Fanuc TP program (LS listing): ground_truth.ls

/PROG  TOR_XL_LEARN_V6
/ATTR
OWNER		= MNEDITOR;
COMMENT		= "WeldPRO Auto-Gen";
PROG_SIZE	= 7125;
CREATE		= DATE 26-07-31  TIME 09:44:06;
MODIFIED	= DATE 26-07-31  TIME 10:09:20;
FILE_NAME	= TOR_XL_L;
VERSION		= 0;
LINE_COUNT	= 113;
MEMORY_SIZE	= 7445;
PROTECT		= READ_WRITE;
TCD:  STACK_SIZE	= 0,
      TASK_PRIORITY	= 50,
      TIME_SLICE	= 0,
      BUSY_LAMP_OFF	= 0,
      ABORT_REQUEST	= 0,
      PAUSE_REQUEST	= 0;
DEFAULT_GROUP	= 1,*,*,*,*;
CONTROL_CODE	= 00000000 00000000;
/APPL
/MN
   1:  !WeldPRO Auto-Generated TPP ;
   2:  !TOR_XL_2026, TOR_xl_2907 ;
   3:   ;
   4:  UFRAME_NUM=2 ;
   5:  UTOOL_NUM=2 ;
   6:  !Feature Approach ;
   7:J P[1]{
   GP1:
	UF : 2, UT : 2,		CONFIG : 'F D T, 0, 0, 0',
	X =   924.335  mm,	Y =   780.986  mm,	Z =  -268.284  mm,
	W =  -106.495 deg,	P =   -15.000 deg,	R =    94.234 deg
};
P[2]{
   GP1:
	UF : 2, UT : 2,		CONFIG : 'F D T, 0, 0, 0',
	X =  1019.644  mm,	Y =   781.684  mm,	Z =  -244.550  mm,
	W =  -106.499 deg,	P =   -14.997 deg,	R =    94.226 deg
};
P[3]{
   GP1:
	UF : 2, UT : 2,		CONFIG : 'F D T, 0, 0, 0',
	X =  1020.405  mm,	Y =   799.754  mm,	Z =  -244.462  mm,
	W =  -106.481 deg,	P =   -15.218 deg,	R =    85.605 deg
};
P[4]{
   GP1:
	UF : 2, UT : 2,		CONFIG : 'F D T, 0, 0, 0',
	X =  1021.641  mm,	Y =   809.652  mm,	Z =  -244.272  mm,
	W =  -106.456 deg,	P =   -15.335 deg,	R =    80.815 deg
};
P[5]{
   GP1:
	UF : 2, UT : 2,		CONFIG : 'F D T, 0, 0, 0',
	X =  1024.226  mm,	Y =   819.374  mm,	Z =  -244.379  mm,
	W =  -106.423 deg,	P =   -15.450 deg,	R =    76.090 deg
};
P[6]{
   GP1:
	UF : 2, UT : 2,		CONFIG : 'F D T, 0, 0, 0',
	X =  1027.311  mm,	Y =   828.945  mm,	Z =  -244.649  mm,
	W =  -106.378 deg,	P =   -15.565 deg,	R =    71.217 deg
};
P[7]{
   GP1:
	UF : 2, UT : 2,		CONFIG : 'F D T, 0, 0, 0',
	X =  1030.979  mm,	Y =   838.150  mm,	Z =  -244.447  mm,
	W =  -106.322 deg,	P =   -15.679 deg,	R =    66.207 deg
};
P[8]{
   GP1:
	UF : 2, UT : 2,		CONFIG : 'F D T, 0, 0, 0',
	X =  1035.354  mm,	Y =   847.225  mm,	Z =  -244.816  mm,
	W =  -106.254 deg,	P =   -15.791 deg,	R =    61.015 deg
};
P[9]{
   GP1:
	UF : 2, UT : 2,		CONFIG : 'F D T, 0, 0, 0',
	X =  1040.784  mm,	Y =   855.509  mm,	Z =  -244.591  mm,
	W =  -106.177 deg,	P =   -15.894 deg,	R =    55.979 deg
};
P[10]{
   GP1:
	UF : 2, UT : 2,		CONFIG : 'F D T, 0, 0, 0',
	X =  1046.817  mm,	Y =   863.336  mm,	Z =  -244.346  mm,
	W =  -106.096 deg,	P =   -15.986 deg,	R =    51.162 deg
};
P[11]{
   GP1:
	UF : 2, UT : 2,		CONFIG : 'F D T, 0, 0, 0',
	X =  1052.848  mm,	Y =   870.760  mm,	Z =  -242.978  mm,
	W =  -106.012 deg,	P =   -16.066 deg,	R =    46.632 deg
};
P[12]{
   GP1:
	UF : 2, UT : 2,		CONFIG : 'F D T, 0, 0, 0',
	X =  1060.411  mm,	Y =   877.610  mm,	Z =  -243.849  mm,
	W =  -105.919 deg,	P =   -16.142 deg,	R =    41.952 deg
};
P[13]{
   GP1:
	UF : 2, UT : 2,		CONFIG : 'F D T, 0, 0, 0',
	X =  1068.135  mm,	Y =   883.678  mm,	Z =  -243.271  mm,
	W =  -105.870 deg,	P =   -16.177 deg,	R =    39.609 deg
};
P[14]{
   GP1:
	UF : 2, UT : 2,		CONFIG : 'F D T, 0, 0, 0',
	X =  1075.871  mm,	Y =   889.554  mm,	Z =  -242.602  mm,
	W =  -105.777 deg,	P =   -16.235 deg,	R =    35.365 deg
};
P[15]{
   GP1:
	UF : 2, UT : 2,		CONFIG : 'F D T, 0, 0, 0',
	X =  1084.231  mm,	Y =   894.951  mm,	Z =  -242.749  mm,
	W =  -105.677 deg,	P =   -16.289 deg,	R =    30.964 deg
};
P[16]{
   GP1:
	UF : 2, UT : 2,		CONFIG : 'F D T, 0, 0, 0',
	X =  1092.767  mm,	Y =   899.377  mm,	Z =  -241.733  mm,
	W =  -105.579 deg,	P =   -16.333 deg,	R =    26.830 deg
};
P[17]{
   GP1:
	UF : 2, UT : 2,		CONFIG : 'F D T, 0, 0, 0',
	X =  1101.511  mm,	Y =   903.615  mm,	Z =  -240.969  mm,
	W =  -105.536 deg,	P =   -16.344 deg,	R =    25.018 deg
};
P[18]{
   GP1:
	UF : 2, UT : 2,		CONFIG : 'F D T, 0, 0, 0',
	X =  1110.599  mm,	Y =   907.764  mm,	Z =  -240.204  mm,
	W =  -116.027 deg,	P =   -16.063 deg,	R =    30.267 deg
};
P[19]{
   GP1:
	UF : 2, UT : 2,		CONFIG : 'F D T, 0, 0, 0',
	X =  1119.110  mm,	Y =   911.431  mm,	Z =  -237.438  mm,
	W =  -126.877 deg,	P =   -15.356 deg,	R =    25.893 deg
};
P[20]{
   GP1:
	UF : 2, UT : 2,		CONFIG : 'F D T, 0, 0, 0',
	X =  1124.636  mm,	Y =   915.856  mm,	Z =  -231.569  mm,
	W =  -119.393 deg,	P =   -15.981 deg,	R =    16.221 deg
};
P[21]{
   GP1:
	UF : 2, UT : 2,		CONFIG : 'F D T, 0, 0, 0',
	X =  1130.332  mm,	Y =   918.277  mm,	Z =  -223.769  mm,
	W =  -115.329 deg,	P =   -16.208 deg,	R =    11.788 deg
};
P[22]{
   GP1:
	UF : 2, UT : 2,		CONFIG : 'F D T, 0, 0, 0',
	X =  1135.965  mm,	Y =   920.698  mm,	Z =  -215.261  mm,
	W =  -112.639 deg,	P =   -16.315 deg,	R =     9.714 deg
};
P[23]{
   GP1:
	UF : 2, UT : 2,		CONFIG : 'F D T, 0, 0, 0',
	X =  1142.866  mm,	Y =   922.459  mm,	Z =  -207.612  mm,
	W =  -110.015 deg,	P =   -16.386 deg,	R =     9.649 deg
};
P[24]{
   GP1:
	UF : 2, UT : 2,		CONFIG : 'F D T, 0, 0, 0',
	X =  1147.332  mm,	Y =   922.394  mm,	Z =  -203.438  mm,
	W =  -108.552 deg,	P =   -16.418 deg,	R =     8.950 deg
};
P[25]{
   GP1:
	UF : 2, UT : 2,		CONFIG : 'F D T, 0, 0, 0',
	X =  1160.590  mm,	Y =   924.719  mm,	Z =  -199.064  mm,
	W =  -105.409 deg,	P =   -16.443 deg,	R =     6.805 deg
};
P[26]{
   GP1:
	UF : 2, UT : 2,		CONFIG : 'F D T, 0, 0, 0',
	X =  1170.242  mm,	Y =   925.769  mm,	Z =  -198.137  mm,
	W =  -104.866 deg,	P =   -16.444 deg,	R =     5.597 deg
};
P[27]{
   GP1:
	UF : 2, UT : 2,		CONFIG : 'F D T, 0, 0, 0',
	X =  1179.912  mm,	Y =   926.392  mm,	Z =  -197.642  mm,
	W =  -104.887 deg,	P =   -16.444 deg,	R =     3.523 deg
};
P[28]{
   GP1:
	UF : 2, UT : 2,		CONFIG : 'F D T, 0, 0, 0',
	X =  1189.521  mm,	Y =   926.618  mm,	Z =  -197.414  mm,
	W =  -104.930 deg,	P =   -16.439 deg,	R =     -.729 deg
};
P[29]{
   GP1:
	UF : 2, UT : 2,		CONFIG : 'F D T, 0, 0, 0',
	X =  1198.921  mm,	Y =   925.996  mm,	Z =  -196.698  mm,
	W =  -104.979 deg,	P =   -16.424 deg,	R =    -5.541 deg
};
P[30]{
   GP1:
	UF : 2, UT : 2,		CONFIG : 'F D T, 0, 0, 0',
	X =  1208.360  mm,	Y =   924.432  mm,	Z =  -196.495  mm,
	W =  -105.028 deg,	P =   -16.400 deg,	R =   -10.259 deg
};
P[31]{
   GP1:
	UF : 2, UT : 2,		CONFIG : 'F D T, 0, 0, 0',
	X =  1217.503  mm,	Y =   922.249  mm,	Z =  -195.799  mm,
	W =  -105.070 deg,	P =   -16.371 deg,	R =   -14.490 deg
};
P[32]{
   GP1:
	UF : 2, UT : 2,		CONFIG : 'F D T, 0, 0, 0',
	X =  1226.788  mm,	Y =   919.719  mm,	Z =  -195.521  mm,
	W =  -105.112 deg,	P =   -16.334 deg,	R =   -18.515 deg
};
P[33]{
   GP1:
	UF : 2, UT : 2,		CONFIG : 'F D T, 0, 0, 0',
	X =  1235.541  mm,	Y =   915.921  mm,	Z =  -195.278  mm,
	W =  -105.158 deg,	P =   -16.285 deg,	R =   -23.051 deg
};
P[34]{
   GP1:
	UF : 2, UT : 2,		CONFIG : 'F D T, 0, 0, 0',
	X =  1243.913  mm,	Y =   912.024  mm,	Z =  -194.613  mm,
	W =  -105.219 deg,	P =   -16.204 deg,	R =   -29.417 deg
};
P[35]{
   GP1:
	UF : 2, UT : 2,		CONFIG : 'F D T, 0, 0, 0',
	X =  1258.745  mm,	Y =   900.651  mm,	Z =  -193.238  mm,
	W =  -105.307 deg,	P =   -16.055 deg,	R =   -38.974 deg
};
P[36]{
   GP1:
	UF : 2, UT : 2,		CONFIG : 'F D T, 0, 0, 0',
	X =  1266.264  mm,	Y =   894.270  mm,	Z =  -192.829  mm,
	W =  -105.302 deg,	P =   -16.063 deg,	R =   -38.625 deg
};
P[37]{
   GP1:
	UF : 2, UT : 2,		CONFIG : 'F D T, 0, 0, 0',
	X =  1273.637  mm,	Y =   888.618  mm,	Z =  -192.422  mm,
	W =  -105.469 deg,	P =   -15.944 deg,	R =   -44.976 deg
};
P[38]{
   GP1:
	UF : 2, UT : 2,		CONFIG : 'F D T, 0, 0, 0',
	X =  1280.382  mm,	Y =   881.861  mm,	Z =  -192.421  mm,
	W =  -105.661 deg,	P =   -15.890 deg,	R =   -47.714 deg
};
P[39]{
   GP1:
	UF : 2, UT : 2,		CONFIG : 'F D T, 0, 0, 0',
	X =  1287.172  mm,	Y =   875.257  mm,	Z =  -193.053  mm,
	W =  -106.210 deg,	P =   -15.792 deg,	R =   -52.259 deg
};
P[40]{
   GP1:
	UF : 2, UT : 2,		CONFIG : 'F D T, 0, 0, 0',
	X =  1293.618  mm,	Y =   868.274  mm,	Z =  -193.889  mm,
	W =  -106.927 deg,	P =   -15.688 deg,	R =   -56.663 deg
};
P[41]{
   GP1:
	UF : 2, UT : 2,		CONFIG : 'F D T, 0, 0, 0',
	X =  1299.152  mm,	Y =   860.597  mm,	Z =  -194.716  mm,
	W =  -107.603 deg,	P =   -15.597 deg,	R =   -60.243 deg
};
P[42]{
   GP1:
	UF : 2, UT : 2,		CONFIG : 'F D T, 0, 0, 0',
	X =  1303.253  mm,	Y =   852.111  mm,	Z =  -195.594  mm,
	W =  -108.271 deg,	P =   -15.504 deg,	R =   -63.685 deg
};
P[43]{
   GP1:
	UF : 2, UT : 2,		CONFIG : 'F D T, 0, 0, 0',
	X =  1307.637  mm,	Y =   843.537  mm,	Z =  -197.369  mm,
	W =  -109.144 deg,	P =   -15.377 deg,	R =   -68.203 deg
};
P[44]{
   GP1:
	UF : 2, UT : 2,		CONFIG : 'F D T, 0, 0, 0',
	X =  1311.234  mm,	Y =   834.808  mm,	Z =  -198.159  mm,
	W =  -109.899 deg,	P =   -15.253 deg,	R =   -72.505 deg
};
P[45]{
   GP1:
	UF : 2, UT : 2,		CONFIG : 'F D T, 0, 0, 0',
	X =  1315.584  mm,	Y =   825.679  mm,	Z =  -200.220  mm,
	W =  -110.273 deg,	P =   -15.181 deg,	R =   -74.981 deg
};
P[46]{
   GP1:
	UF : 2, UT : 2,		CONFIG : 'F D T, 0, 0, 0',
	X =  1317.524  mm,	Y =   815.957  mm,	Z =  -200.846  mm,
	W =  -110.635 deg,	P =   -14.305 deg,	R =   -78.232 deg
};
P[47]{
   GP1:
	UF : 2, UT : 2,		CONFIG : 'F D T, 0, 0, 0',
	X =  1318.740  mm,	Y =   806.239  mm,	Z =  -201.928  mm,
	W =  -111.054 deg,	P =   -14.769 deg,	R =   -83.164 deg
};
P[48]{
   GP1:
	UF : 2, UT : 2,		CONFIG : 'F D T, 0, 0, 0',
	X =  1320.516  mm,	Y =   796.409  mm,	Z =  -202.991  mm,
	W =  -111.190 deg,	P =   -15.305 deg,	R =   -88.308 deg
};
P[49]{
   GP1:
	UF : 2, UT : 2,		CONFIG : 'F D T, 0, 0, 0',
	X =  1320.184  mm,	Y =   786.553  mm,	Z =  -202.824  mm,
	W =  -111.129 deg,	P =   -15.645 deg,	R =   -91.614 deg
};
P[50]{
   GP1:
	UF : 2, UT : 2,		CONFIG : 'F D T, 0, 0, 0',
	X =  1320.238  mm,	Y =   776.295  mm,	Z =  -202.567  mm,
	W =  -110.757 deg,	P =   -14.624 deg,	R =   -96.575 deg
};
P[51]{
   GP1:
	UF : 2, UT : 2,		CONFIG : 'F D T, 0, 0, 0',
	X =  1318.522  mm,	Y =   766.566  mm,	Z =  -201.487  mm,
	W =  -110.276 deg,	P =   -14.535 deg,	R =  -100.836 deg
};
P[52]{
   GP1:
	UF : 2, UT : 2,		CONFIG : 'F D T, 0, 0, 0',
	X =  1317.605  mm,	Y =   756.550  mm,	Z =  -200.428  mm,
	W =  -109.635 deg,	P =   -14.447 deg,	R =  -105.265 deg
};
P[53]{
   GP1:
	UF : 2, UT : 2,		CONFIG : 'F D T, 0, 0, 0',
	X =  1315.114  mm,	Y =   746.859  mm,	Z =  -199.251  mm,
	W =  -109.083 deg,	P =   -14.382 deg,	R =  -108.625 deg
};
P[54]{
   GP1:
	UF : 2, UT : 2,		CONFIG : 'F D T, 0, 0, 0',
	X =  1311.521  mm,	Y =   737.672  mm,	Z =  -197.517  mm,
	W =  -108.349 deg,	P =   -14.302 deg,	R =  -112.873 deg
};
P[55]{
   GP1:
	UF : 2, UT : 2,		CONFIG : 'F D T, 0, 0, 0',
	X =  1307.398  mm,	Y =   728.719  mm,	Z =  -195.709  mm,
	W =  -107.748 deg,	P =   -14.239 deg,	R =  -116.265 deg
};
P[56]{
   GP1:
	UF : 2, UT : 2,		CONFIG : 'F D T, 0, 0, 0',
	X =  1303.277  mm,	Y =   719.710  mm,	Z =  -194.166  mm,
	W =  -106.924 deg,	P =   -14.148 deg,	R =  -121.191 deg
};
P[57]{
   GP1:
	UF : 2, UT : 2,		CONFIG : 'F D T, 0, 0, 0',
	X =  1298.077  mm,	Y =   711.301  mm,	Z =  -192.670  mm,
	W =  -106.269 deg,	P =   -14.066 deg,	R =  -125.698 deg
};
P[58]{
   GP1:
	UF : 2, UT : 2,		CONFIG : 'F D T, 0, 0, 0',
	X =  1292.024  mm,	Y =   703.662  mm,	Z =  -190.774  mm,
	W =  -105.781 deg,	P =   -13.988 deg,	R =  -130.143 deg
};
P[59]{
   GP1:
	UF : 2, UT : 2,		CONFIG : 'F D T, 0, 0, 0',
	X =  1285.800  mm,	Y =   695.686  mm,	Z =  -190.310  mm,
	W =  -105.527 deg,	P =   -13.913 deg,	R =  -134.519 deg
};
P[60]{
   GP1:
	UF : 2, UT : 2,		CONFIG : 'F D T, 0, 0, 0',
	X =  1279.455  mm,	Y =   688.076  mm,	Z =  -189.451  mm,
	W =  -105.437 deg,	P =   -13.849 deg,	R =  -138.629 deg
};
P[61]{
   GP1:
	UF : 2, UT : 2,		CONFIG : 'F D T, 0, 0, 0',
	X =  1272.079  mm,	Y =   681.121  mm,	Z =  -189.791  mm,
	W =  -105.429 deg,	P =   -13.831 deg,	R =  -139.837 deg
};
P[62]{
   GP1:
	UF : 2, UT : 2,		CONFIG : 'F D T, 0, 0, 0',
	X =  1264.269  mm,	Y =   675.069  mm,	Z =  -189.390  mm,
	W =  -105.443 deg,	P =   -13.863 deg,	R =  -137.727 deg
};
P[63]{
   GP1:
	UF : 2, UT : 2,		CONFIG : 'F D T, 0, 0, 0',
	X =  1256.776  mm,	Y =   667.526  mm,	Z =  -190.522  mm,
	W =  -105.373 deg,	P =   -13.729 deg,	R =  -147.436 deg
};
P[64]{
   GP1:
	UF : 2, UT : 2,		CONFIG : 'F D T, 0, 0, 0',
	X =  1248.434  mm,	Y =   660.897  mm,	Z =  -190.873  mm,
	W =  -105.298 deg,	P =   -13.637 deg,	R =  -156.529 deg
};
P[65]{
   GP1:
	UF : 2, UT : 2,		CONFIG : 'F D T, 0, 0, 0',
	X =  1239.073  mm,	Y =   657.015  mm,	Z =  -190.882  mm,
	W =  -105.277 deg,	P =   -13.618 deg,	R =  -158.976 deg
};
P[66]{
   GP1:
	UF : 2, UT : 2,		CONFIG : 'F D T, 0, 0, 0',
	X =  1229.501  mm,	Y =   653.024  mm,	Z =  -191.408  mm,
	W =  -105.241 deg,	P =   -13.592 deg,	R =  -162.969 deg
};
P[67]{
   GP1:
	UF : 2, UT : 2,		CONFIG : 'F D T, 0, 0, 0',
	X =  1219.671  mm,	Y =   649.816  mm,	Z =  -191.704  mm,
	W =  -105.203 deg,	P =   -13.573 deg,	R =  -167.022 deg
};
P[68]{
   GP1:
	UF : 2, UT : 2,		CONFIG : 'F D T, 0, 0, 0',
	X =  1209.583  mm,	Y =   647.190  mm,	Z =  -192.082  mm,
	W =  -105.159 deg,	P =   -13.560 deg,	R =  -171.569 deg
};
P[69]{
   GP1:
	UF : 2, UT : 2,		CONFIG : 'F D T, 0, 0, 0',
	X =  1199.122  mm,	Y =   646.053  mm,	Z =  -192.900  mm,
	W =  -105.113 deg,	P =   -13.556 deg,	R =  -176.312 deg
};
P[70]{
   GP1:
	UF : 2, UT : 2,		CONFIG : 'F D T, 0, 0, 0',
	X =  1188.683  mm,	Y =   645.625  mm,	Z =  -193.481  mm,
	W =  -105.068 deg,	P =   -13.561 deg,	R =   179.213 deg
};
P[71]{
   GP1:
	UF : 2, UT : 2,		CONFIG : 'F D T, 0, 0, 0',
	X =  1178.492  mm,	Y =   646.246  mm,	Z =  -193.489  mm,
	W =  -105.038 deg,	P =   -13.569 deg,	R =   176.231 deg
};
P[72]{
   GP1:
	UF : 2, UT : 2,		CONFIG : 'F D T, 0, 0, 0',
	X =  1168.209  mm,	Y =   647.153  mm,	Z =  -194.575  mm,
	W =  -105.207 deg,	P =   -13.572 deg,	R =   175.290 deg
};
P[73]{
   GP1:
	UF : 2, UT : 2,		CONFIG : 'F D T, 0, 0, 0',
	X =  1158.558  mm,	Y =   647.646  mm,	Z =  -195.439  mm,
	W =  -107.012 deg,	P =   -13.569 deg,	R =   174.537 deg
};
P[74]{
   GP1:
	UF : 2, UT : 2,		CONFIG : 'F D T, 0, 0, 0',
	X =  1149.794  mm,	Y =   648.269  mm,	Z =  -198.347  mm,
	W =  -109.414 deg,	P =   -13.538 deg,	R =   174.483 deg
};
P[75]{
   GP1:
	UF : 2, UT : 2,		CONFIG : 'F D T, 0, 0, 0',
	X =  1142.506  mm,	Y =   649.272  mm,	Z =  -202.713  mm,
	W =  -112.196 deg,	P =   -13.466 deg,	R =   175.323 deg
};
P[76]{
   GP1:
	UF : 2, UT : 2,		CONFIG : 'F D T, 0, 0, 0',
	X =  1136.383  mm,	Y =   650.304  mm,	Z =  -209.368  mm,
	W =  -114.872 deg,	P =   -13.369 deg,	R =   175.422 deg
};
P[77]{
   GP1:
	UF : 2, UT : 2,		CONFIG : 'F D T, 0, 0, 0',
	X =  1129.205  mm,	Y =   652.569  mm,	Z =  -220.097  mm,
	W =  -120.114 deg,	P =   -13.109 deg,	R =   172.293 deg
};
P[78]{
   GP1:
	UF : 2, UT : 2,		CONFIG : 'F D T, 0, 0, 0',
	X =  1122.221  mm,	Y =   656.579  mm,	Z =  -230.126  mm,
	W =  -126.809 deg,	P =   -12.620 deg,	R =   167.792 deg
};
P[79]{
   GP1:
	UF : 2, UT : 2,		CONFIG : 'F D T, 0, 0, 0',
	X =  1113.460  mm,	Y =   661.332  mm,	Z =  -235.426  mm,
	W =  -119.561 deg,	P =   -13.285 deg,	R =   157.806 deg
};
P[80]{
   GP1:
	UF : 2, UT : 2,		CONFIG : 'F D T, 0, 0, 0',
	X =  1103.909  mm,	Y =   665.641  mm,	Z =  -237.067  mm,
	W =  -107.219 deg,	P =   -13.741 deg,	R =   154.408 deg
};
P[81]{
   GP1:
	UF : 2, UT : 2,		CONFIG : 'F D T, 0, 0, 0',
	X =  1094.631  mm,	Y =   669.875  mm,	Z =  -237.862  mm,
	W =  -105.746 deg,	P =   -13.749 deg,	R =   154.142 deg
};
P[82]{
   GP1:
	UF : 2, UT : 2,		CONFIG : 'F D T, 0, 0, 0',
	X =  1085.640  mm,	Y =   675.021  mm,	Z =  -238.534  mm,
	W =  -105.804 deg,	P =   -13.784 deg,	R =   151.506 deg
};
P[83]{
   GP1:
	UF : 2, UT : 2,		CONFIG : 'F D T, 0, 0, 0',
	X =  1076.501  mm,	Y =   680.297  mm,	Z =  -239.671  mm,
	W =  -105.885 deg,	P =   -13.838 deg,	R =   147.739 deg
};
P[84]{
   GP1:
	UF : 2, UT : 2,		CONFIG : 'F D T, 0, 0, 0',
	X =  1067.906  mm,	Y =   686.478  mm,	Z =  -240.491  mm,
	W =  -105.988 deg,	P =   -13.918 deg,	R =   142.681 deg
};
P[85]{
   GP1:
	UF : 2, UT : 2,		CONFIG : 'F D T, 0, 0, 0',
	X =  1060.318  mm,	Y =   693.668  mm,	Z =  -240.705  mm,
	W =  -106.084 deg,	P =   -14.001 deg,	R =   137.677 deg
};
P[86]{
   GP1:
	UF : 2, UT : 2,		CONFIG : 'F D T, 0, 0, 0',
	X =  1053.073  mm,	Y =   700.857  mm,	Z =  -241.184  mm,
	W =  -106.129 deg,	P =   -14.056 deg,	R =   135.015 deg
};
P[87]{
   GP1:
	UF : 2, UT : 2,		CONFIG : 'F D T, 0, 0, 0',
	X =  1046.171  mm,	Y =   708.523  mm,	Z =  -241.638  mm,
	W =  -106.186 deg,	P =   -14.117 deg,	R =   131.622 deg
};
P[88]{
   GP1:
	UF : 2, UT : 2,		CONFIG : 'F D T, 0, 0, 0',
	X =  1039.540  mm,	Y =   716.621  mm,	Z =  -242.396  mm,
	W =  -106.269 deg,	P =   -14.239 deg,	R =   125.999 deg
};
P[89]{
   GP1:
	UF : 2, UT : 2,		CONFIG : 'F D T, 0, 0, 0',
	X =  1034.197  mm,	Y =   725.380  mm,	Z =  -242.834  mm,
	W =  -106.343 deg,	P =   -14.367 deg,	R =   120.225 deg
};
P[90]{
   GP1:
	UF : 2, UT : 2,		CONFIG : 'F D T, 0, 0, 0',
	X =  1030.258  mm,	Y =   733.864  mm,	Z =  -243.102  mm,
	W =  -106.383 deg,	P =   -14.448 deg,	R =   116.672 deg
};
P[91]{
   GP1:
	UF : 2, UT : 2,		CONFIG : 'F D T, 0, 0, 0',
	X =  1025.999  mm,	Y =   742.170  mm,	Z =  -243.646  mm,
	W =  -106.433 deg,	P =   -14.556 deg,	R =   111.957 deg
};
P[92]{
   GP1:
	UF : 2, UT : 2,		CONFIG : 'F D T, 0, 0, 0',
	X =  1023.110  mm,	Y =   754.360  mm,	Z =  -244.123  mm,
	W =  -106.465 deg,	P =   -14.714 deg,	R =   105.666 deg
};
P[93]{
   GP1:
	UF : 2, UT : 2,		CONFIG : 'F D T, 0, 1, 0',
	X =  1020.432  mm,	Y =   764.197  mm,	Z =  -244.429  mm,
	W =  -106.480 deg,	P =   -14.798 deg,	R =   102.261 deg
};
P[94]{
   GP1:
	UF : 2, UT : 2,		CONFIG : 'F D T, 0, 0, 0',
	X =  1014.789  mm,	Y =   776.665  mm,	Z =  -227.278  mm,
	W =  -106.497 deg,	P =   -14.995 deg,	R =    94.216 deg
};
P[95]{
   GP1:
	UF : 2, UT : 2,		CONFIG : 'F D T, 0, 1, 0',
	X =  1019.376  mm,	Y =   774.295  mm,	Z =  -244.242  mm,
	W =  -106.494 deg,	P =   -14.935 deg,	R =    96.827 deg
};
P[96]{
   GP1:
	UF : 2, UT : 2,		CONFIG : 'F D T, 0, 1, 0',
	X =  1018.860  mm,	Y =   781.671  mm,	Z =  -244.718  mm,
	W =  -106.501 deg,	P =   -15.000 deg,	R =    94.236 deg
};
P[97]{
   GP1:
	UF : 2, UT : 2,		CONFIG : 'F D T, 0, 0, 0',
	X =  1020.164  mm,	Y =   789.679  mm,	Z =  -244.298  mm,
	W =  -106.492 deg,	P =   -15.098 deg,	R =    90.372 deg
};
P[98]{
   GP1:
	UF : 2, UT : 2,		CONFIG : 'F D T, 0, 1, 0',
	X =   651.995  mm,	Y =   781.694  mm,	Z =  -345.952  mm,
	W =  -106.495 deg,	P =   -15.000 deg,	R =    94.234 deg
};

/END
